FUNCTION_BLOCK FB_FunctionCompositionCustomized
VAR
	count	: INT	:= 0;
	TTAZone : ST_ZoneData;
	latch	: BOOL := FALSE;
END_VAR

//fbF_10_001_0200_02_0.CtrlIn.DestinationFunction := F_10_001_0230_01_0;
//fbF_10_001_0200_02_0.CtrlIn.DestinationZone := 1;
//fbF_10_001_0200_02_0.CtrlIn.TU_Type := 1;

//fbF_10_001_0200_02_0.CtrlIn.DestinationFunction := F_10_001_0215_01_0;
//fbF_10_001_0200_02_0.CtrlIn.DestinationZone := 2;
//fbF_10_001_0200_02_0.CtrlIn.TU_Type := 1;

TTAZone := F_GetZoneData(E_FunctionNumber.F_10_001_0200_01_0, 1);
IF NOT TTAZone.TransportControlData.Occupied THEN
IF count = 0 AND NOT latch THEN 
	fbF_10_001_0200_02_0.CtrlIn.DestinationFunction := F_10_001_0233_01_0;
	fbF_10_001_0200_02_0.CtrlIn.DestinationZone := 1;
	fbF_10_001_0200_02_0.CtrlIn.TU_Type := 1;
	count := count + 1;
	latch := TRUE;
ELSIF count = 1 AND NOT latch THEN
	fbF_10_001_0200_02_0.CtrlIn.DestinationFunction := F_10_001_0215_01_0;
	fbF_10_001_0200_02_0.CtrlIn.DestinationZone := 2;
	fbF_10_001_0200_02_0.CtrlIn.TU_Type := 1;
	count := count + 1;
	latch := TRUE;
ELSIF count = 2 AND NOT latch THEN
	fbF_10_001_0200_02_0.CtrlIn.DestinationFunction := F_10_001_0213_01_0;
	fbF_10_001_0200_02_0.CtrlIn.DestinationZone := 1;
	fbF_10_001_0200_02_0.CtrlIn.TU_Type := 1;
	count := count + 1;
	latch := TRUE;
ELSIF count = 3 AND NOT latch THEN
	fbF_10_001_0200_02_0.CtrlIn.DestinationFunction := F_10_001_0207_01_0;
	fbF_10_001_0200_02_0.CtrlIn.DestinationZone := 1;
	fbF_10_001_0200_02_0.CtrlIn.TU_Type := 1;
	count := count + 1;
	latch := TRUE;
ELSIF count = 4 AND NOT latch THEN
	fbF_10_001_0200_02_0.CtrlIn.DestinationFunction := F_10_001_0232_01_0;
	fbF_10_001_0200_02_0.CtrlIn.DestinationZone := 1;
	fbF_10_001_0200_02_0.CtrlIn.TU_Type := 1;
	count := 0;
	latch := TRUE;
END_IF
ELSE 
	latch := FALSE;
END_IF

END_FUNCTION_BLOCK

(* stored: Version 1.1.0.1, ProductVersion 3.1.4024.9
   POU FB_FunctionCompositionCustomized: Id {dab6032a-07a7-4e89-86c7-4672b3b39b9a}, SpecialFunc None *)
